Fanuc KAREL source: NC0045.KL

-- PROVISIONAL review KL for V940-1; original PC SHA256 10b29d344562ec8dd383c79f34a4f856aac042b55be89b65df79f98c66e7d979
-- Incomplete behavior may be omitted. Consult companion uncertainty JSON. Do not deploy.
PROGRAM NC0045
%NOLOCKGROUP
-- UNRESOLVED_LOCAL_POOL 1 cells at code offset 3; source declarations unknown
-- DIRECT_LOCAL_WORD_ACCESS alone does not prove INTEGER, REAL, or BOOLEAN
BEGIN
  -- V9_CONDITION_STACK_HINT 3 bounded expression windows; static native code-base-relative target link; source arms held
  -- UNRESOLVED_PC offsets 0-8; opcodes 2B,2C,7B
  -- UNRESOLVED_PC offsets 13-20; opcodes 9D,23
  -- UNRESOLVED_PC offsets 25-38; opcodes 21,9D,57,79
  -- UNRESOLVED_PC offsets 43-60; opcodes 21,40,41,42
  -- UNRESOLVED_PC offsets 65-78; opcodes 21,9D,57,79
  -- UNRESOLVED_PC offsets 83-100; opcodes 21,40,41,42
  -- UNRESOLVED_PC offsets 105-118; opcodes 21,9D,57,79
  -- UNRESOLVED_PC offsets 123-137; opcodes 21,9D,52,23
  -- UNRESOLVED_PC offsets 142-147; opcodes 7A
  -- UNRESOLVED_PC offsets 152-170; opcodes 21,2E,52,23
  -- UNRESOLVED_PC offsets 175-191; opcodes 7A,40,41,42
  -- UNRESOLVED_PC offsets 196-220; opcodes 21,2E,52,23,7A,43
  -- UNRESOLVED_PC offsets 225-243; opcodes 21,2E,52,23
  -- UNRESOLVED_PC offsets 253-258; opcodes 7A
  -- UNRESOLVED_PC offsets 263-281; opcodes 21,2E,52,23
  -- UNRESOLVED_PC offsets 286-302; opcodes 7A,40,41,42
  -- UNRESOLVED_PC offsets 307-331; opcodes 21,2E,52,23,7A,43
  -- UNRESOLVED_PC offsets 336-354; opcodes 21,2E,52,23
  -- UNRESOLVED_PC offsets 364-369; opcodes 7A
  -- UNRESOLVED_PC offsets 374-392; opcodes 21,2E,52,23
  -- UNRESOLVED_PC offsets 402-406; opcodes 7F
  -- UNRESOLVED_PC offsets 411-415; opcodes 27,AA
  -- UNRESOLVED_PC offsets 420-424; opcodes 7F
END NC0045
